// TIA Portal project "Control PID de nivel_V20" (V20)

(* hardware
DEVICE "Estación S7-1500/ET200MP_1"  S7-1500 station
   slot 0: "Perfil soporte_0"  Rack  6ES7 590-1***0-0AA0
   slot 1: "PLC_1"  CPU 1511-1 PN  6ES7 511-1AK02-0AB0  V2.9
      slot 3: "Display de la CPU_1"  6ES7591-1AA00-0AA0
      slot 32768: "Interfaz PROFINET_1"  X1
         slot 32769: "Puerto_1"  X1 P1
         slot 32770: "Puerto_2"  X1 P2
      slot 34817: "Virtual CP interface port_1"  Virtual CP interface port  Virtual CP interface port
*)

// ===== PLC "PLC_1"  CPU 1511-1 PN =====

VAR_GLOBAL   // PLC tag table "Tabla de variables estándar"
   "Level meter" AT %ID100 : Real;
   "Flow meter" AT %ID104 : Real;
   "Setpoint" AT %ID108 : Real;
   "Fill valve" AT %QD100 : Real;
   "Regularlor Salida" AT %ID112 : Real;
   "SP" AT %QD108 : DInt;
   "PV" AT %QD112 : DInt;
   "Clock_Byte" AT %MB9998 : Byte;
   "Clock_10Hz" AT %M9998.0 : Bool;
   "Clock_5Hz" AT %M9998.1 : Bool;
   "Clock_2.5Hz" AT %M9998.2 : Bool;
   "Clock_2Hz" AT %M9998.3 : Bool;
   "Clock_1.25Hz" AT %M9998.4 : Bool;
   "Clock_1Hz" AT %M9998.5 : Bool;
   "Clock_0.625Hz" AT %M9998.6 : Bool;
   "Clock_0.5Hz" AT %M9998.7 : Bool;
   "System_Byte" AT %MB9999 : Byte;
   "FirstScan" AT %M9999.0 : Bool;
   "DiagStatusUpdate" AT %M9999.1 : Bool;
   "AlwaysTRUE" AT %M9999.2 : Bool;
   "AlwaysFALSE" AT %M9999.3 : Bool;
   "nivel_norm" AT %MD6 : Real;
   "nivel" AT %MD0 : Real;
   "valvula_salida_norm" AT %MD10 : Real;
   "valvula_salida" AT %MD14 : Real;
   "SP_Real" AT %MD18 : Real;
   "manual" AT %M4.0 : Bool;
   "valor manual" AT %MD22 : Real;
   "Nivel Deposito" AT %QD116 : DInt;
   "Valvula Descarga" AT %QD104 : Real;
   "Salida" AT %QD120 : DInt;
   "Regularlor Salida norm" AT %MD26 : Real;
END_VAR

ORGANIZATION_BLOCK "Main"   // OB1, LAD, ProgramCycle
TITLE = "Main Program Sweep (Cycle)"
{ S7_Optimized_Access := 'TRUE' }
VERSION : 0.1
   VAR_INPUT
      Initial_Call : Bool;   // Initial call of this OB
      Remanence : Bool;   // =True, if remanent data are available
   END_VAR
BEGIN

REGION Network 1
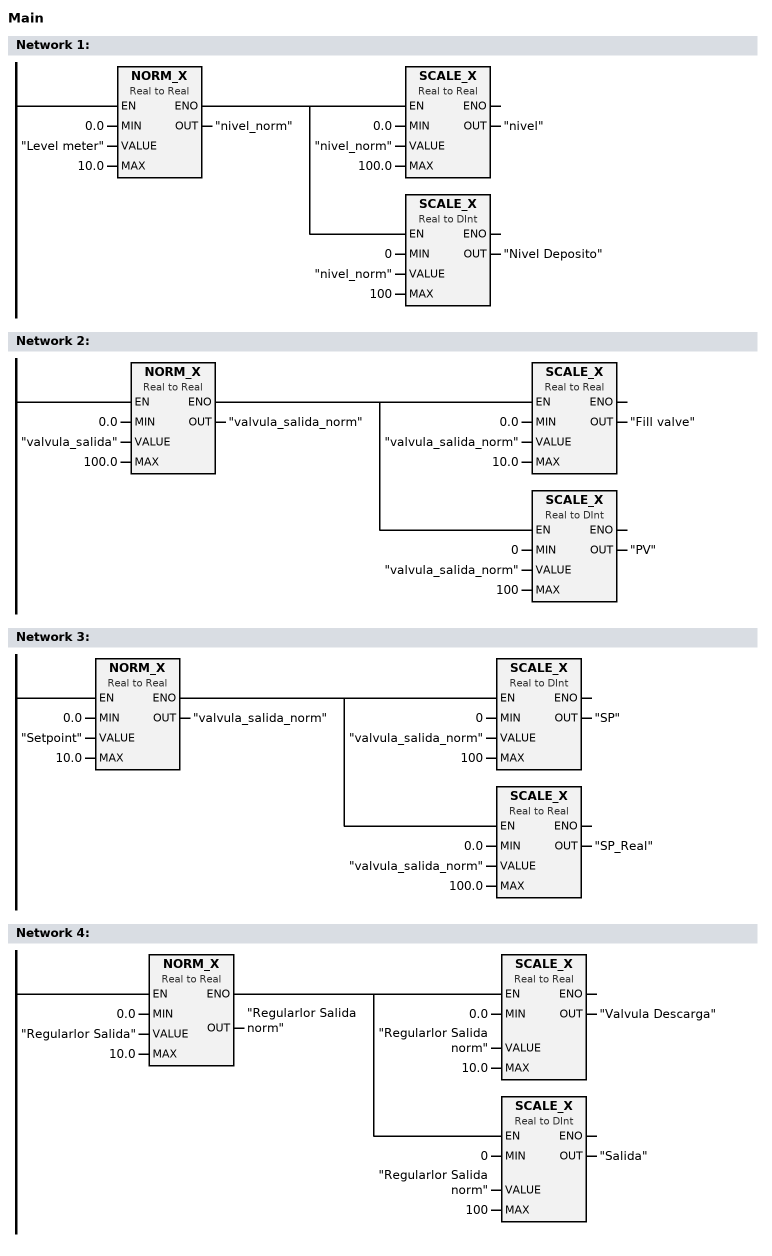
   RUNG wire#powerrail
      { S7_Templates := "[SrcType := Real, DestType := Real]" } Normalize(min := 0.0, value := "Level meter", max := 10.0, out => "nivel_norm")
      wire#w1
      { S7_Templates := "[SrcType := Real, DestType := Real]" } Scale(min := 0.0, value := "nivel_norm", max := 100.0, out => "nivel")
   END_RUNG
   RUNG wire#w1
      { S7_Templates := "[SrcType := Real, DestType := DInt]" } Scale(min := 0, value := "nivel_norm", max := 100, out => "Nivel Deposito")
   END_RUNG
   // the same network as SCL:
   "nivel_norm" := NORM_X(MIN := 0.0, VALUE := "Level meter", MAX := 10.0);
   "nivel" := SCALE_X(MIN := 0.0, VALUE := "nivel_norm", MAX := 100.0);
   "Nivel Deposito" := SCALE_X(MIN := 0, VALUE := "nivel_norm", MAX := 100);
END_REGION

REGION Network 2
   RUNG wire#powerrail
      { S7_Templates := "[SrcType := Real, DestType := Real]" } Normalize(min := 0.0, value := "valvula_salida", max := 100.0, out => "valvula_salida_norm")
      wire#w1
      { S7_Templates := "[SrcType := Real, DestType := Real]" } Scale(min := 0.0, value := "valvula_salida_norm", max := 10.0, out => "Fill valve")
   END_RUNG
   RUNG wire#w1
      { S7_Templates := "[SrcType := Real, DestType := DInt]" } Scale(min := 0, value := "valvula_salida_norm", max := 100, out => "PV")
   END_RUNG
   // the same network as SCL:
   "valvula_salida_norm" := NORM_X(MIN := 0.0, VALUE := "valvula_salida", MAX := 100.0);
   "Fill valve" := SCALE_X(MIN := 0.0, VALUE := "valvula_salida_norm", MAX := 10.0);
   "PV" := SCALE_X(MIN := 0, VALUE := "valvula_salida_norm", MAX := 100);
END_REGION

REGION Network 3
   RUNG wire#powerrail
      { S7_Templates := "[SrcType := Real, DestType := Real]" } Normalize(min := 0.0, value := "Setpoint", max := 10.0, out => "valvula_salida_norm")
      wire#w1
      { S7_Templates := "[SrcType := Real, DestType := DInt]" } Scale(min := 0, value := "valvula_salida_norm", max := 100, out => "SP")
   END_RUNG
   RUNG wire#w1
      { S7_Templates := "[SrcType := Real, DestType := Real]" } Scale(min := 0.0, value := "valvula_salida_norm", max := 100.0, out => "SP_Real")
   END_RUNG
   // the same network as SCL:
   "valvula_salida_norm" := NORM_X(MIN := 0.0, VALUE := "Setpoint", MAX := 10.0);
   "SP" := SCALE_X(MIN := 0, VALUE := "valvula_salida_norm", MAX := 100);
   "SP_Real" := SCALE_X(MIN := 0.0, VALUE := "valvula_salida_norm", MAX := 100.0);
END_REGION

REGION Network 4
   RUNG wire#powerrail
      { S7_Templates := "[SrcType := Real, DestType := Real]" } Normalize(min := 0.0, value := "Regularlor Salida", max := 10.0, out => "Regularlor Salida norm")
      wire#w1
      { S7_Templates := "[SrcType := Real, DestType := Real]" } Scale(min := 0.0, value := "Regularlor Salida norm", max := 10.0, out => "Valvula Descarga")
   END_RUNG
   RUNG wire#w1
      { S7_Templates := "[SrcType := Real, DestType := DInt]" } Scale(min := 0, value := "Regularlor Salida norm", max := 100, out => "Salida")
   END_RUNG
   // the same network as SCL:
   "Regularlor Salida norm" := NORM_X(MIN := 0.0, VALUE := "Regularlor Salida", MAX := 10.0);
   "Valvula Descarga" := SCALE_X(MIN := 0.0, VALUE := "Regularlor Salida norm", MAX := 10.0);
   "Salida" := SCALE_X(MIN := 0, VALUE := "Regularlor Salida norm", MAX := 100);
END_REGION
END_ORGANIZATION_BLOCK

ORGANIZATION_BLOCK "Cyclic interrupt"   // OB30, LAD, CyclicInterrupt
{ S7_Optimized_Access := 'TRUE' }
VERSION : 0.1
   VAR_INPUT
      Initial_Call : Bool;   // Initial call of this OB
      Event_Count : Int;   // Events discarded
   END_VAR
BEGIN

REGION Network 1
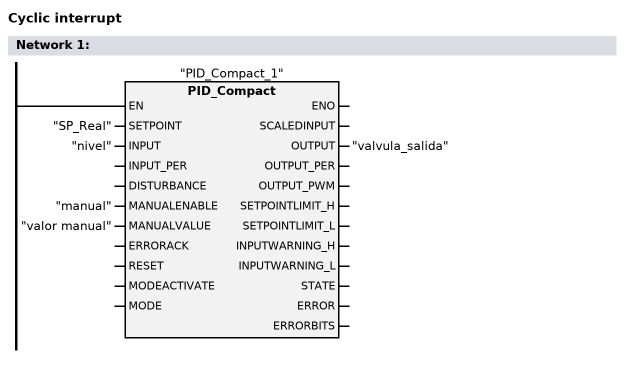
   "PID_Compact_1"(Setpoint := "SP_Real",   // PID_Compact
                   Input := "nivel",
                   ManualEnable := "manual",
                   ManualValue := "valor manual",
                   Output => "valvula_salida");
END_REGION
END_ORGANIZATION_BLOCK